    Lines7[76].X := 237.960; Lines7[76].Z := 284.913; Lines7[76].F := 800; Lines7[76].CMD := 1; Lines7[76].Param := 0; // G1 Linear [Op11 P1]
    Lines7[77].X := 237.085; Lines7[77].Z := 286.141; Lines7[77].F := 800; Lines7[77].CMD := 1; Lines7[77].Param := 0; // G1 Linear [Op11 P1]
    Lines7[78].X := 236.206; Lines7[78].Z := 287.367; Lines7[78].F := 800; Lines7[78].CMD := 1; Lines7[78].Param := 0; // G1 Linear [Op11 P1]
    Lines7[79].X := 235.321; Lines7[79].Z := 288.589; Lines7[79].F := 800; Lines7[79].CMD := 1; Lines7[79].Param := 0; // G1 Linear [Op11 P1]
    Lines7[80].X := 234.432; Lines7[80].Z := 289.808; Lines7[80].F := 800; Lines7[80].CMD := 1; Lines7[80].Param := 0; // G1 Linear [Op11 P1]
    Lines7[81].X := 233.539; Lines7[81].Z := 291.025; Lines7[81].F := 800; Lines7[81].CMD := 1; Lines7[81].Param := 0; // G1 Linear [Op11 P1]
    Lines7[82].X := 232.491; Lines7[82].Z := 292.440; Lines7[82].F := 800; Lines7[82].CMD := 1; Lines7[82].Param := 0; // G1 Linear [Op11 P1]
    Lines7[83].X := 231.587; Lines7[83].Z := 293.650; Lines7[83].F := 800; Lines7[83].CMD := 1; Lines7[83].Param := 0; // G1 Linear [Op11 P1]
    Lines7[84].X := 230.678; Lines7[84].Z := 294.858; Lines7[84].F := 800; Lines7[84].CMD := 1; Lines7[84].Param := 0; // G1 Linear [Op11 P1]
    Lines7[85].X := 229.765; Lines7[85].Z := 296.062; Lines7[85].F := 800; Lines7[85].CMD := 1; Lines7[85].Param := 0; // G1 Linear [Op11 P1]
    Lines7[86].X := 228.848; Lines7[86].Z := 297.263; Lines7[86].F := 800; Lines7[86].CMD := 1; Lines7[86].Param := 0; // G1 Linear [Op11 P1]
    Lines7[87].X := 227.925; Lines7[87].Z := 298.462; Lines7[87].F := 800; Lines7[87].CMD := 1; Lines7[87].Param := 0; // G1 Linear [Op11 P1]
    Lines7[88].X := 226.843; Lines7[88].Z := 299.857; Lines7[88].F := 800; Lines7[88].CMD := 1; Lines7[88].Param := 0; // G1 Linear [Op11 P1]
    Lines7[89].X := 225.911; Lines7[89].Z := 301.049; Lines7[89].F := 800; Lines7[89].CMD := 1; Lines7[89].Param := 0; // G1 Linear [Op11 P1]
    Lines7[90].X := 224.974; Lines7[90].Z := 302.238; Lines7[90].F := 800; Lines7[90].CMD := 1; Lines7[90].Param := 0; // G1 Linear [Op11 P1]
    Lines7[91].X := 224.032; Lines7[91].Z := 303.424; Lines7[91].F := 800; Lines7[91].CMD := 1; Lines7[91].Param := 0; // G1 Linear [Op11 P1]
    Lines7[92].X := 222.927; Lines7[92].Z := 304.805; Lines7[92].F := 800; Lines7[92].CMD := 1; Lines7[92].Param := 0; // G1 Linear [Op11 P1]
    Lines7[93].X := 212.927; Lines7[93].Z := 294.805; Lines7[93].F := 0; Lines7[93].CMD := 0; Lines7[93].Param := 0; // G0 Rapid [Op11 P1]
    Lines7[94].X := 212.927; Lines7[94].Z := 294.805; Lines7[94].F := 0; Lines7[94].CMD := 20; Lines7[94].Param := 80; // Spindle ON 800 RPM [Op11 P1]
    Lines7[95].X := 275.949; Lines7[95].Z := 196.000; Lines7[95].F := 0; Lines7[95].CMD := 0; Lines7[95].Param := 0; // G0 Rapid [Op12 P1]
    Lines7[96].X := 275.844; Lines7[96].Z := 227.468; Lines7[96].F := 800; Lines7[96].CMD := 1; Lines7[96].Param := 0; // G1 Linear [Op12 P1]
    Lines7[97].X := 275.813; Lines7[97].Z := 227.813; Lines7[97].F := 800; Lines7[97].CMD := 1; Lines7[97].Param := 0; // G1 Linear [Op12 P1]
    Lines7[98].X := 275.723; Lines7[98].Z := 228.147; Lines7[98].F := 800; Lines7[98].CMD := 1; Lines7[98].Param := 0; // G1 Linear [Op12 P1]
    Lines7[99].X := 275.576; Lines7[99].Z := 228.461; Lines7[99].F := 800; Lines7[99].CMD := 1; Lines7[99].Param := 0; // G1 Linear [Op12 P1]
    Lines8[0].X := 274.987; Lines8[0].Z := 229.860; Lines8[0].F := 800; Lines8[0].CMD := 1; Lines8[0].Param := 0; // G1 Linear [Op12 P1]
    Lines8[1].X := 274.392; Lines8[1].Z := 231.257; Lines8[1].F := 800; Lines8[1].CMD := 1; Lines8[1].Param := 0; // G1 Linear [Op12 P1]
    Lines8[2].X := 273.287; Lines8[2].Z := 233.809; Lines8[2].F := 800; Lines8[2].CMD := 1; Lines8[2].Param := 0; // G1 Linear [Op12 P1]
    Lines8[3].X := 272.677; Lines8[3].Z := 235.197; Lines8[3].F := 800; Lines8[3].CMD := 1; Lines8[3].Param := 0; // G1 Linear [Op12 P1]
    Lines8[4].X := 272.062; Lines8[4].Z := 236.582; Lines8[4].F := 800; Lines8[4].CMD := 1; Lines8[4].Param := 0; // G1 Linear [Op12 P1]
    Lines8[5].X := 271.441; Lines8[5].Z := 237.964; Lines8[5].F := 800; Lines8[5].CMD := 1; Lines8[5].Param := 0; // G1 Linear [Op12 P1]
    Lines8[6].X := 270.815; Lines8[6].Z := 239.343; Lines8[6].F := 800; Lines8[6].CMD := 1; Lines8[6].Param := 0; // G1 Linear [Op12 P1]
    Lines8[7].X := 269.654; Lines8[7].Z := 241.863; Lines8[7].F := 800; Lines8[7].CMD := 1; Lines8[7].Param := 0; // G1 Linear [Op12 P1]
    Lines8[8].X := 269.013; Lines8[8].Z := 243.233; Lines8[8].F := 800; Lines8[8].CMD := 1; Lines8[8].Param := 0; // G1 Linear [Op12 P1]
    Lines8[9].X := 268.367; Lines8[9].Z := 244.600; Lines8[9].F := 800; Lines8[9].CMD := 1; Lines8[9].Param := 0; // G1 Linear [Op12 P1]
    Lines8[10].X := 267.716; Lines8[10].Z := 245.964; Lines8[10].F := 800; Lines8[10].CMD := 1; Lines8[10].Param := 0; // G1 Linear [Op12 P1]
    Lines8[11].X := 267.059; Lines8[11].Z := 247.325; Lines8[11].F := 800; Lines8[11].CMD := 1; Lines8[11].Param := 0; // G1 Linear [Op12 P1]
    Lines8[12].X := 266.397; Lines8[12].Z := 248.683; Lines8[12].F := 800; Lines8[12].CMD := 1; Lines8[12].Param := 0; // G1 Linear [Op12 P1]
    Lines8[13].X := 265.729; Lines8[13].Z := 250.038; Lines8[13].F := 800; Lines8[13].CMD := 1; Lines8[13].Param := 0; // G1 Linear [Op12 P1]
    Lines8[14].X := 264.492; Lines8[14].Z := 252.514; Lines8[14].F := 800; Lines8[14].CMD := 1; Lines8[14].Param := 0; // G1 Linear [Op12 P1]
    Lines8[15].X := 263.810; Lines8[15].Z := 253.860; Lines8[15].F := 800; Lines8[15].CMD := 1; Lines8[15].Param := 0; // G1 Linear [Op12 P1]
    Lines8[16].X := 263.122; Lines8[16].Z := 255.203; Lines8[16].F := 800; Lines8[16].CMD := 1; Lines8[16].Param := 0; // G1 Linear [Op12 P1]
    Lines8[17].X := 262.429; Lines8[17].Z := 256.543; Lines8[17].F := 800; Lines8[17].CMD := 1; Lines8[17].Param := 0; // G1 Linear [Op12 P1]
    Lines8[18].X := 261.731; Lines8[18].Z := 257.880; Lines8[18].F := 800; Lines8[18].CMD := 1; Lines8[18].Param := 0; // G1 Linear [Op12 P1]
    Lines8[19].X := 261.027; Lines8[19].Z := 259.214; Lines8[19].F := 800; Lines8[19].CMD := 1; Lines8[19].Param := 0; // G1 Linear [Op12 P1]
    Lines8[20].X := 260.319; Lines8[20].Z := 260.545; Lines8[20].F := 800; Lines8[20].CMD := 1; Lines8[20].Param := 0; // G1 Linear [Op12 P1]
    Lines8[21].X := 259.005; Lines8[21].Z := 262.977; Lines8[21].F := 800; Lines8[21].CMD := 1; Lines8[21].Param := 0; // G1 Linear [Op12 P1]
    Lines8[22].X := 258.282; Lines8[22].Z := 264.300; Lines8[22].F := 800; Lines8[22].CMD := 1; Lines8[22].Param := 0; // G1 Linear [Op12 P1]
    Lines8[23].X := 257.552; Lines8[23].Z := 265.619; Lines8[23].F := 800; Lines8[23].CMD := 1; Lines8[23].Param := 0; // G1 Linear [Op12 P1]
    Lines8[24].X := 256.818; Lines8[24].Z := 266.935; Lines8[24].F := 800; Lines8[24].CMD := 1; Lines8[24].Param := 0; // G1 Linear [Op12 P1]
    Lines8[25].X := 256.078; Lines8[25].Z := 268.248; Lines8[25].F := 800; Lines8[25].CMD := 1; Lines8[25].Param := 0; // G1 Linear [Op12 P1]
    Lines8[26].X := 255.333; Lines8[26].Z := 269.558; Lines8[26].F := 800; Lines8[26].CMD := 1; Lines8[26].Param := 0; // G1 Linear [Op12 P1]
    Lines8[27].X := 254.583; Lines8[27].Z := 270.865; Lines8[27].F := 800; Lines8[27].CMD := 1; Lines8[27].Param := 0; // G1 Linear [Op12 P1]
    Lines8[28].X := 253.827; Lines8[28].Z := 272.169; Lines8[28].F := 800; Lines8[28].CMD := 1; Lines8[28].Param := 0; // G1 Linear [Op12 P1]
    Lines8[29].X := 253.067; Lines8[29].Z := 273.470; Lines8[29].F := 800; Lines8[29].CMD := 1; Lines8[29].Param := 0; // G1 Linear [Op12 P1]
    Lines8[30].X := 252.300; Lines8[30].Z := 274.768; Lines8[30].F := 800; Lines8[30].CMD := 1; Lines8[30].Param := 0; // G1 Linear [Op12 P1]
    Lines8[31].X := 251.529; Lines8[31].Z := 276.063; Lines8[31].F := 800; Lines8[31].CMD := 1; Lines8[31].Param := 0; // G1 Linear [Op12 P1]
    Lines8[32].X := 250.752; Lines8[32].Z := 277.355; Lines8[32].F := 800; Lines8[32].CMD := 1; Lines8[32].Param := 0; // G1 Linear [Op12 P1]
    Lines8[33].X := 249.970; Lines8[33].Z := 278.643; Lines8[33].F := 800; Lines8[33].CMD := 1; Lines8[33].Param := 0; // G1 Linear [Op12 P1]
    Lines8[34].X := 248.523; Lines8[34].Z := 280.998; Lines8[34].F := 800; Lines8[34].CMD := 1; Lines8[34].Param := 0; // G1 Linear [Op12 P1]
    Lines8[35].X := 247.057; Lines8[35].Z := 283.343; Lines8[35].F := 800; Lines8[35].CMD := 1; Lines8[35].Param := 0; // G1 Linear [Op12 P1]
    Lines8[36].X := 246.250; Lines8[36].Z := 284.617; Lines8[36].F := 800; Lines8[36].CMD := 1; Lines8[36].Param := 0; // G1 Linear [Op12 P1]
    Lines8[37].X := 245.438; Lines8[37].Z := 285.888; Lines8[37].F := 800; Lines8[37].CMD := 1; Lines8[37].Param := 0; // G1 Linear [Op12 P1]
    Lines8[38].X := 244.621; Lines8[38].Z := 287.157; Lines8[38].F := 800; Lines8[38].CMD := 1; Lines8[38].Param := 0; // G1 Linear [Op12 P1]
    Lines8[39].X := 243.798; Lines8[39].Z := 288.422; Lines8[39].F := 800; Lines8[39].CMD := 1; Lines8[39].Param := 0; // G1 Linear [Op12 P1]
    Lines8[40].X := 242.971; Lines8[40].Z := 289.684; Lines8[40].F := 800; Lines8[40].CMD := 1; Lines8[40].Param := 0; // G1 Linear [Op12 P1]
    Lines8[41].X := 242.137; Lines8[41].Z := 290.944; Lines8[41].F := 800; Lines8[41].CMD := 1; Lines8[41].Param := 0; // G1 Linear [Op12 P1]
    Lines8[42].X := 240.596; Lines8[42].Z := 293.244; Lines8[42].F := 800; Lines8[42].CMD := 1; Lines8[42].Param := 0; // G1 Linear [Op12 P1]
    Lines8[43].X := 239.748; Lines8[43].Z := 294.495; Lines8[43].F := 800; Lines8[43].CMD := 1; Lines8[43].Param := 0; // G1 Linear [Op12 P1]
    Lines8[44].X := 238.894; Lines8[44].Z := 295.742; Lines8[44].F := 800; Lines8[44].CMD := 1; Lines8[44].Param := 0; // G1 Linear [Op12 P1]
    Lines8[45].X := 238.035; Lines8[45].Z := 296.987; Lines8[45].F := 800; Lines8[45].CMD := 1; Lines8[45].Param := 0; // G1 Linear [Op12 P1]
    Lines8[46].X := 237.171; Lines8[46].Z := 298.228; Lines8[46].F := 800; Lines8[46].CMD := 1; Lines8[46].Param := 0; // G1 Linear [Op12 P1]
    Lines8[47].X := 236.302; Lines8[47].Z := 299.466; Lines8[47].F := 800; Lines8[47].CMD := 1; Lines8[47].Param := 0; // G1 Linear [Op12 P1]
    Lines8[48].X := 235.427; Lines8[48].Z := 300.702; Lines8[48].F := 800; Lines8[48].CMD := 1; Lines8[48].Param := 0; // G1 Linear [Op12 P1]
    Lines8[49].X := 234.547; Lines8[49].Z := 301.934; Lines8[49].F := 800; Lines8[49].CMD := 1; Lines8[49].Param := 0; // G1 Linear [Op12 P1]
    Lines8[50].X := 233.662; Lines8[50].Z := 303.163; Lines8[50].F := 800; Lines8[50].CMD := 1; Lines8[50].Param := 0; // G1 Linear [Op12 P1]
    Lines8[51].X := 232.025; Lines8[51].Z := 305.409; Lines8[51].F := 800; Lines8[51].CMD := 1; Lines8[51].Param := 0; // G1 Linear [Op12 P1]
    Lines8[52].X := 231.125; Lines8[52].Z := 306.629; Lines8[52].F := 800; Lines8[52].CMD := 1; Lines8[52].Param := 0; // G1 Linear [Op12 P1]
    Lines8[53].X := 230.219; Lines8[53].Z := 307.847; Lines8[53].F := 800; Lines8[53].CMD := 1; Lines8[53].Param := 0; // G1 Linear [Op12 P1]
    Lines8[54].X := 229.308; Lines8[54].Z := 309.061; Lines8[54].F := 800; Lines8[54].CMD := 1; Lines8[54].Param := 0; // G1 Linear [Op12 P1]
    Lines8[55].X := 228.392; Lines8[55].Z := 310.272; Lines8[55].F := 800; Lines8[55].CMD := 1; Lines8[55].Param := 0; // G1 Linear [Op12 P1]
    Lines8[56].X := 218.392; Lines8[56].Z := 300.272; Lines8[56].F := 0; Lines8[56].CMD := 0; Lines8[56].Param := 0; // G0 Rapid [Op12 P1]
    Lines8[57].X := 218.392; Lines8[57].Z := 300.272; Lines8[57].F := 0; Lines8[57].CMD := 20; Lines8[57].Param := 80; // Spindle ON 800 RPM [Op12 P1]
    Lines8[58].X := 275.949; Lines8[58].Z := 196.000; Lines8[58].F := 0; Lines8[58].CMD := 0; Lines8[58].Param := 0; // G0 Rapid [Op13 P1]
    Lines8[59].X := 275.819; Lines8[59].Z := 235.000; Lines8[59].F := 400; Lines8[59].CMD := 1; Lines8[59].Param := 0; // G1 Linear [Op13 P1]
    Lines8[60].X := 274.979; Lines8[60].Z := 237.394; Lines8[60].F := 400; Lines8[60].CMD := 1; Lines8[60].Param := 0; // G1 Linear [Op13 P1]
    Lines8[61].X := 274.552; Lines8[61].Z := 238.587; Lines8[61].F := 400; Lines8[61].CMD := 1; Lines8[61].Param := 0; // G1 Linear [Op13 P1]
    Lines8[62].X := 274.034; Lines8[62].Z := 240.016; Lines8[62].F := 400; Lines8[62].CMD := 1; Lines8[62].Param := 0; // G1 Linear [Op13 P1]
    Lines8[63].X := 273.597; Lines8[63].Z := 241.204; Lines8[63].F := 400; Lines8[63].CMD := 1; Lines8[63].Param := 0; // G1 Linear [Op13 P1]
    Lines8[64].X := 273.067; Lines8[64].Z := 242.627; Lines8[64].F := 400; Lines8[64].CMD := 1; Lines8[64].Param := 0; // G1 Linear [Op13 P1]
    Lines8[65].X := 272.621; Lines8[65].Z := 243.811; Lines8[65].F := 400; Lines8[65].CMD := 1; Lines8[65].Param := 0; // G1 Linear [Op13 P1]
    Lines8[66].X := 272.079; Lines8[66].Z := 245.228; Lines8[66].F := 400; Lines8[66].CMD := 1; Lines8[66].Param := 0; // G1 Linear [Op13 P1]
    Lines8[67].X := 271.623; Lines8[67].Z := 246.406; Lines8[67].F := 400; Lines8[67].CMD := 1; Lines8[67].Param := 0; // G1 Linear [Op13 P1]
    Lines8[68].X := 271.070; Lines8[68].Z := 247.817; Lines8[68].F := 400; Lines8[68].CMD := 1; Lines8[68].Param := 0; // G1 Linear [Op13 P1]
    Lines8[69].X := 270.510; Lines8[69].Z := 249.225; Lines8[69].F := 400; Lines8[69].CMD := 1; Lines8[69].Param := 0; // G1 Linear [Op13 P1]
    Lines8[70].X := 270.038; Lines8[70].Z := 250.396; Lines8[70].F := 400; Lines8[70].CMD := 1; Lines8[70].Param := 0; // G1 Linear [Op13 P1]
    Lines8[71].X := 269.563; Lines8[71].Z := 251.564; Lines8[71].F := 400; Lines8[71].CMD := 1; Lines8[71].Param := 0; // G1 Linear [Op13 P1]
    Lines8[72].X := 268.986; Lines8[72].Z := 252.963; Lines8[72].F := 400; Lines8[72].CMD := 1; Lines8[72].Param := 0; // G1 Linear [Op13 P1]
    Lines8[73].X := 268.010; Lines8[73].Z := 255.288; Lines8[73].F := 400; Lines8[73].CMD := 1; Lines8[73].Param := 0; // G1 Linear [Op13 P1]
    Lines8[74].X := 267.515; Lines8[74].Z := 256.447; Lines8[74].F := 400; Lines8[74].CMD := 1; Lines8[74].Param := 0; // G1 Linear [Op13 P1]
    Lines8[75].X := 266.915; Lines8[75].Z := 257.834; Lines8[75].F := 400; Lines8[75].CMD := 1; Lines8[75].Param := 0; // G1 Linear [Op13 P1]
    Lines8[76].X := 266.411; Lines8[76].Z := 258.988; Lines8[76].F := 400; Lines8[76].CMD := 1; Lines8[76].Param := 0; // G1 Linear [Op13 P1]
    Lines8[77].X := 265.800; Lines8[77].Z := 260.370; Lines8[77].F := 400; Lines8[77].CMD := 1; Lines8[77].Param := 0; // G1 Linear [Op13 P1]
    Lines8[78].X := 265.285; Lines8[78].Z := 261.518; Lines8[78].F := 400; Lines8[78].CMD := 1; Lines8[78].Param := 0; // G1 Linear [Op13 P1]
    Lines8[79].X := 264.662; Lines8[79].Z := 262.894; Lines8[79].F := 400; Lines8[79].CMD := 1; Lines8[79].Param := 0; // G1 Linear [Op13 P1]
    Lines8[80].X := 264.033; Lines8[80].Z := 264.266; Lines8[80].F := 400; Lines8[80].CMD := 1; Lines8[80].Param := 0; // G1 Linear [Op13 P1]
    Lines8[81].X := 263.503; Lines8[81].Z := 265.408; Lines8[81].F := 400; Lines8[81].CMD := 1; Lines8[81].Param := 0; // G1 Linear [Op13 P1]
    Lines8[82].X := 262.969; Lines8[82].Z := 266.546; Lines8[82].F := 400; Lines8[82].CMD := 1; Lines8[82].Param := 0; // G1 Linear [Op13 P1]
    Lines8[83].X := 262.322; Lines8[83].Z := 267.910; Lines8[83].F := 400; Lines8[83].CMD := 1; Lines8[83].Param := 0; // G1 Linear [Op13 P1]
    Lines8[84].X := 261.779; Lines8[84].Z := 269.044; Lines8[84].F := 400; Lines8[84].CMD := 1; Lines8[84].Param := 0; // G1 Linear [Op13 P1]
    Lines8[85].X := 261.120; Lines8[85].Z := 270.401; Lines8[85].F := 400; Lines8[85].CMD := 1; Lines8[85].Param := 0; // G1 Linear [Op13 P1]
    Lines8[86].X := 260.008; Lines8[86].Z := 272.657; Lines8[86].F := 400; Lines8[86].CMD := 1; Lines8[86].Param := 0; // G1 Linear [Op13 P1]
    Lines8[87].X := 259.446; Lines8[87].Z := 273.781; Lines8[87].F := 400; Lines8[87].CMD := 1; Lines8[87].Param := 0; // G1 Linear [Op13 P1]
    Lines8[88].X := 258.765; Lines8[88].Z := 275.127; Lines8[88].F := 400; Lines8[88].CMD := 1; Lines8[88].Param := 0; // G1 Linear [Op13 P1]
    Lines8[89].X := 257.616; Lines8[89].Z := 277.364; Lines8[89].F := 400; Lines8[89].CMD := 1; Lines8[89].Param := 0; // G1 Linear [Op13 P1]
    Lines8[90].X := 257.034; Lines8[90].Z := 278.478; Lines8[90].F := 400; Lines8[90].CMD := 1; Lines8[90].Param := 0; // G1 Linear [Op13 P1]
    Lines8[91].X := 256.331; Lines8[91].Z := 279.813; Lines8[91].F := 400; Lines8[91].CMD := 1; Lines8[91].Param := 0; // G1 Linear [Op13 P1]
    Lines8[92].X := 255.621; Lines8[92].Z := 281.144; Lines8[92].F := 400; Lines8[92].CMD := 1; Lines8[92].Param := 0; // G1 Linear [Op13 P1]
    Lines8[93].X := 255.024; Lines8[93].Z := 282.251; Lines8[93].F := 400; Lines8[93].CMD := 1; Lines8[93].Param := 0; // G1 Linear [Op13 P1]
    Lines8[94].X := 254.423; Lines8[94].Z := 283.356; Lines8[94].F := 400; Lines8[94].CMD := 1; Lines8[94].Param := 0; // G1 Linear [Op13 P1]
    Lines8[95].X := 253.696; Lines8[95].Z := 284.679; Lines8[95].F := 400; Lines8[95].CMD := 1; Lines8[95].Param := 0; // G1 Linear [Op13 P1]
    Lines8[96].X := 252.470; Lines8[96].Z := 286.876; Lines8[96].F := 400; Lines8[96].CMD := 1; Lines8[96].Param := 0; // G1 Linear [Op13 P1]
    Lines8[97].X := 251.726; Lines8[97].Z := 288.190; Lines8[97].F := 400; Lines8[97].CMD := 1; Lines8[97].Param := 0; // G1 Linear [Op13 P1]
    Lines8[98].X := 251.101; Lines8[98].Z := 289.282; Lines8[98].F := 400; Lines8[98].CMD := 1; Lines8[98].Param := 0; // G1 Linear [Op13 P1]
    Lines8[99].X := 250.471; Lines8[99].Z := 290.373; Lines8[99].F := 400; Lines8[99].CMD := 1; Lines8[99].Param := 0; // G1 Linear [Op13 P1]
    Lines9[0].X := 249.710; Lines9[0].Z := 291.678; Lines9[0].F := 400; Lines9[0].CMD := 1; Lines9[0].Param := 0; // G1 Linear [Op13 P1]
    Lines9[1].X := 249.071; Lines9[1].Z := 292.763; Lines9[1].F := 400; Lines9[1].CMD := 1; Lines9[1].Param := 0; // G1 Linear [Op13 P1]
    Lines9[2].X := 248.297; Lines9[2].Z := 294.062; Lines9[2].F := 400; Lines9[2].CMD := 1; Lines9[2].Param := 0; // G1 Linear [Op13 P1]
    Lines9[3].X := 246.995; Lines9[3].Z := 296.220; Lines9[3].F := 400; Lines9[3].CMD := 1; Lines9[3].Param := 0; // G1 Linear [Op13 P1]
    Lines9[4].X := 246.336; Lines9[4].Z := 297.296; Lines9[4].F := 400; Lines9[4].CMD := 1; Lines9[4].Param := 0; // G1 Linear [Op13 P1]
    Lines9[5].X := 245.541; Lines9[5].Z := 298.584; Lines9[5].F := 400; Lines9[5].CMD := 1; Lines9[5].Param := 0; // G1 Linear [Op13 P1]
    Lines9[6].X := 244.873; Lines9[6].Z := 299.654; Lines9[6].F := 400; Lines9[6].CMD := 1; Lines9[6].Param := 0; // G1 Linear [Op13 P1]
    Lines9[7].X := 244.065; Lines9[7].Z := 300.936; Lines9[7].F := 400; Lines9[7].CMD := 1; Lines9[7].Param := 0; // G1 Linear [Op13 P1]
    Lines9[8].X := 243.387; Lines9[8].Z := 302.002; Lines9[8].F := 400; Lines9[8].CMD := 1; Lines9[8].Param := 0; // G1 Linear [Op13 P1]
    Lines9[9].X := 242.568; Lines9[9].Z := 303.278; Lines9[9].F := 400; Lines9[9].CMD := 1; Lines9[9].Param := 0; // G1 Linear [Op13 P1]
    Lines9[10].X := 241.881; Lines9[10].Z := 304.338; Lines9[10].F := 400; Lines9[10].CMD := 1; Lines9[10].Param := 0; // G1 Linear [Op13 P1]
    Lines9[11].X := 241.049; Lines9[11].Z := 305.608; Lines9[11].F := 400; Lines9[11].CMD := 1; Lines9[11].Param := 0; // G1 Linear [Op13 P1]
    Lines9[12].X := 240.352; Lines9[12].Z := 306.664; Lines9[12].F := 400; Lines9[12].CMD := 1; Lines9[12].Param := 0; // G1 Linear [Op13 P1]
    Lines9[13].X := 239.509; Lines9[13].Z := 307.927; Lines9[13].F := 400; Lines9[13].CMD := 1; Lines9[13].Param := 0; // G1 Linear [Op13 P1]
    Lines9[14].X := 238.802; Lines9[14].Z := 308.978; Lines9[14].F := 400; Lines9[14].CMD := 1; Lines9[14].Param := 0; // G1 Linear [Op13 P1]
    Lines9[15].X := 237.947; Lines9[15].Z := 310.236; Lines9[15].F := 400; Lines9[15].CMD := 1; Lines9[15].Param := 0; // G1 Linear [Op13 P1]
    Lines9[16].X := 237.230; Lines9[16].Z := 311.281; Lines9[16].F := 400; Lines9[16].CMD := 1; Lines9[16].Param := 0; // G1 Linear [Op13 P1]
    Lines9[17].X := 236.364; Lines9[17].Z := 312.533; Lines9[17].F := 400; Lines9[17].CMD := 1; Lines9[17].Param := 0; // G1 Linear [Op13 P1]
    Lines9[18].X := 226.364; Lines9[18].Z := 302.533; Lines9[18].F := 0; Lines9[18].CMD := 0; Lines9[18].Param := 0; // G0 Rapid [Op13 P1]
    Lines9[19].X := 226.364; Lines9[19].Z := 302.533; Lines9[19].F := 0; Lines9[19].CMD := 20; Lines9[19].Param := 80; // Spindle ON 800 RPM [Op13 P1]
    Lines9[20].X := 275.882; Lines9[20].Z := 216.000; Lines9[20].F := 0; Lines9[20].CMD := 0; Lines9[20].Param := 0; // G0 Rapid [Op14 P1]
    Lines9[21].X := 275.799; Lines9[21].Z := 241.000; Lines9[21].F := 400; Lines9[21].CMD := 1; Lines9[21].Param := 0; // G1 Linear [Op14 P1]
    Lines9[22].X := 275.441; Lines9[22].Z := 242.217; Lines9[22].F := 400; Lines9[22].CMD := 1; Lines9[22].Param := 0; // G1 Linear [Op14 P1]
    Lines9[23].X := 275.077; Lines9[23].Z := 243.432; Lines9[23].F := 400; Lines9[23].CMD := 1; Lines9[23].Param := 0; // G1 Linear [Op14 P1]
    Lines9[24].X := 274.409; Lines9[24].Z := 245.611; Lines9[24].F := 400; Lines9[24].CMD := 1; Lines9[24].Param := 0; // G1 Linear [Op14 P1]
    Lines9[25].X := 274.030; Lines9[25].Z := 246.818; Lines9[25].F := 400; Lines9[25].CMD := 1; Lines9[25].Param := 0; // G1 Linear [Op14 P1]
    Lines9[26].X := 273.645; Lines9[26].Z := 248.023; Lines9[26].F := 400; Lines9[26].CMD := 1; Lines9[26].Param := 0; // G1 Linear [Op14 P1]
    Lines9[27].X := 273.255; Lines9[27].Z := 249.225; Lines9[27].F := 400; Lines9[27].CMD := 1; Lines9[27].Param := 0; // G1 Linear [Op14 P1]
    Lines9[28].X := 272.859; Lines9[28].Z := 250.424; Lines9[28].F := 400; Lines9[28].CMD := 1; Lines9[28].Param := 0; // G1 Linear [Op14 P1]
    Lines9[29].X := 272.132; Lines9[29].Z := 252.576; Lines9[29].F := 400; Lines9[29].CMD := 1; Lines9[29].Param := 0; // G1 Linear [Op14 P1]
    Lines9[30].X := 271.720; Lines9[30].Z := 253.768; Lines9[30].F := 400; Lines9[30].CMD := 1; Lines9[30].Param := 0; // G1 Linear [Op14 P1]
    Lines9[31].X := 271.303; Lines9[31].Z := 254.958; Lines9[31].F := 400; Lines9[31].CMD := 1; Lines9[31].Param := 0; // G1 Linear [Op14 P1]
    Lines9[32].X := 270.880; Lines9[32].Z := 256.145; Lines9[32].F := 400; Lines9[32].CMD := 1; Lines9[32].Param := 0; // G1 Linear [Op14 P1]
    Lines9[33].X := 270.452; Lines9[33].Z := 257.329; Lines9[33].F := 400; Lines9[33].CMD := 1; Lines9[33].Param := 0; // G1 Linear [Op14 P1]
    Lines9[34].X := 270.018; Lines9[34].Z := 258.511; Lines9[34].F := 400; Lines9[34].CMD := 1; Lines9[34].Param := 0; // G1 Linear [Op14 P1]
    Lines9[35].X := 269.579; Lines9[35].Z := 259.690; Lines9[35].F := 400; Lines9[35].CMD := 1; Lines9[35].Param := 0; // G1 Linear [Op14 P1]
    Lines9[36].X := 268.773; Lines9[36].Z := 261.806; Lines9[36].F := 400; Lines9[36].CMD := 1; Lines9[36].Param := 0; // G1 Linear [Op14 P1]
    Lines9[37].X := 268.318; Lines9[37].Z := 262.977; Lines9[37].F := 400; Lines9[37].CMD := 1; Lines9[37].Param := 0; // G1 Linear [Op14 P1]
    Lines9[38].X := 267.858; Lines9[38].Z := 264.147; Lines9[38].F := 400; Lines9[38].CMD := 1; Lines9[38].Param := 0; // G1 Linear [Op14 P1]
    Lines9[39].X := 267.391; Lines9[39].Z := 265.313; Lines9[39].F := 400; Lines9[39].CMD := 1; Lines9[39].Param := 0; // G1 Linear [Op14 P1]
    Lines9[40].X := 266.919; Lines9[40].Z := 266.477; Lines9[40].F := 400; Lines9[40].CMD := 1; Lines9[40].Param := 0; // G1 Linear [Op14 P1]
    Lines9[41].X := 266.442; Lines9[41].Z := 267.639; Lines9[41].F := 400; Lines9[41].CMD := 1; Lines9[41].Param := 0; // G1 Linear [Op14 P1]
    Lines9[42].X := 265.959; Lines9[42].Z := 268.797; Lines9[42].F := 400; Lines9[42].CMD := 1; Lines9[42].Param := 0; // G1 Linear [Op14 P1]
    Lines9[43].X := 265.075; Lines9[43].Z := 270.877; Lines9[43].F := 400; Lines9[43].CMD := 1; Lines9[43].Param := 0; // G1 Linear [Op14 P1]
    Lines9[44].X := 264.576; Lines9[44].Z := 272.028; Lines9[44].F := 400; Lines9[44].CMD := 1; Lines9[44].Param := 0; // G1 Linear [Op14 P1]
    Lines9[45].X := 264.072; Lines9[45].Z := 273.177; Lines9[45].F := 400; Lines9[45].CMD := 1; Lines9[45].Param := 0; // G1 Linear [Op14 P1]
    Lines9[46].X := 263.562; Lines9[46].Z := 274.323; Lines9[46].F := 400; Lines9[46].CMD := 1; Lines9[46].Param := 0; // G1 Linear [Op14 P1]
    Lines9[47].X := 263.047; Lines9[47].Z := 275.467; Lines9[47].F := 400; Lines9[47].CMD := 1; Lines9[47].Param := 0; // G1 Linear [Op14 P1]
    Lines9[48].X := 262.525; Lines9[48].Z := 276.608; Lines9[48].F := 400; Lines9[48].CMD := 1; Lines9[48].Param := 0; // G1 Linear [Op14 P1]
    Lines9[49].X := 261.999; Lines9[49].Z := 277.747; Lines9[49].F := 400; Lines9[49].CMD := 1; Lines9[49].Param := 0; // G1 Linear [Op14 P1]
    Lines9[50].X := 261.037; Lines9[50].Z := 279.789; Lines9[50].F := 400; Lines9[50].CMD := 1; Lines9[50].Param := 0; // G1 Linear [Op14 P1]
    Lines9[51].X := 260.494; Lines9[51].Z := 280.920; Lines9[51].F := 400; Lines9[51].CMD := 1; Lines9[51].Param := 0; // G1 Linear [Op14 P1]
    Lines9[52].X := 259.946; Lines9[52].Z := 282.049; Lines9[52].F := 400; Lines9[52].CMD := 1; Lines9[52].Param := 0; // G1 Linear [Op14 P1]
    Lines9[53].X := 259.393; Lines9[53].Z := 283.175; Lines9[53].F := 400; Lines9[53].CMD := 1; Lines9[53].Param := 0; // G1 Linear [Op14 P1]
    Lines9[54].X := 258.834; Lines9[54].Z := 284.298; Lines9[54].F := 400; Lines9[54].CMD := 1; Lines9[54].Param := 0; // G1 Linear [Op14 P1]
    Lines9[55].X := 258.269; Lines9[55].Z := 285.419; Lines9[55].F := 400; Lines9[55].CMD := 1; Lines9[55].Param := 0; // G1 Linear [Op14 P1]
    Lines9[56].X := 257.699; Lines9[56].Z := 286.537; Lines9[56].F := 400; Lines9[56].CMD := 1; Lines9[56].Param := 0; // G1 Linear [Op14 P1]
    Lines9[57].X := 257.123; Lines9[57].Z := 287.653; Lines9[57].F := 400; Lines9[57].CMD := 1; Lines9[57].Param := 0; // G1 Linear [Op14 P1]
    Lines9[58].X := 256.542; Lines9[58].Z := 288.766; Lines9[58].F := 400; Lines9[58].CMD := 1; Lines9[58].Param := 0; // G1 Linear [Op14 P1]
    Lines9[59].X := 255.481; Lines9[59].Z := 290.763; Lines9[59].F := 400; Lines9[59].CMD := 1; Lines9[59].Param := 0; // G1 Linear [Op14 P1]
    Lines9[60].X := 254.884; Lines9[60].Z := 291.869; Lines9[60].F := 400; Lines9[60].CMD := 1; Lines9[60].Param := 0; // G1 Linear [Op14 P1]
    Lines9[61].X := 254.281; Lines9[61].Z := 292.972; Lines9[61].F := 400; Lines9[61].CMD := 1; Lines9[61].Param := 0; // G1 Linear [Op14 P1]
    Lines9[62].X := 253.673; Lines9[62].Z := 294.072; Lines9[62].F := 400; Lines9[62].CMD := 1; Lines9[62].Param := 0; // G1 Linear [Op14 P1]
    Lines9[63].X := 253.059; Lines9[63].Z := 295.170; Lines9[63].F := 400; Lines9[63].CMD := 1; Lines9[63].Param := 0; // G1 Linear [Op14 P1]
    Lines9[64].X := 251.940; Lines9[64].Z := 297.140; Lines9[64].F := 400; Lines9[64].CMD := 1; Lines9[64].Param := 0; // G1 Linear [Op14 P1]
    Lines9[65].X := 251.310; Lines9[65].Z := 298.230; Lines9[65].F := 400; Lines9[65].CMD := 1; Lines9[65].Param := 0; // G1 Linear [Op14 P1]
    Lines9[66].X := 250.675; Lines9[66].Z := 299.318; Lines9[66].F := 400; Lines9[66].CMD := 1; Lines9[66].Param := 0; // G1 Linear [Op14 P1]
    Lines9[67].X := 250.035; Lines9[67].Z := 300.404; Lines9[67].F := 400; Lines9[67].CMD := 1; Lines9[67].Param := 0; // G1 Linear [Op14 P1]
    Lines9[68].X := 249.388; Lines9[68].Z := 301.487; Lines9[68].F := 400; Lines9[68].CMD := 1; Lines9[68].Param := 0; // G1 Linear [Op14 P1]
    Lines9[69].X := 248.737; Lines9[69].Z := 302.567; Lines9[69].F := 400; Lines9[69].CMD := 1; Lines9[69].Param := 0; // G1 Linear [Op14 P1]
    Lines9[70].X := 248.079; Lines9[70].Z := 303.644; Lines9[70].F := 400; Lines9[70].CMD := 1; Lines9[70].Param := 0; // G1 Linear [Op14 P1]
    Lines9[71].X := 246.882; Lines9[71].Z := 305.578; Lines9[71].F := 400; Lines9[71].CMD := 1; Lines9[71].Param := 0; // G1 Linear [Op14 P1]
    Lines9[72].X := 246.209; Lines9[72].Z := 306.648; Lines9[72].F := 400; Lines9[72].CMD := 1; Lines9[72].Param := 0; // G1 Linear [Op14 P1]
    Lines9[73].X := 245.530; Lines9[73].Z := 307.716; Lines9[73].F := 400; Lines9[73].CMD := 1; Lines9[73].Param := 0; // G1 Linear [Op14 P1]
    Lines9[74].X := 244.846; Lines9[74].Z := 308.781; Lines9[74].F := 400; Lines9[74].CMD := 1; Lines9[74].Param := 0; // G1 Linear [Op14 P1]
    Lines9[75].X := 244.156; Lines9[75].Z := 309.843; Lines9[75].F := 400; Lines9[75].CMD := 1; Lines9[75].Param := 0; // G1 Linear [Op14 P1]
    Lines9[76].X := 243.460; Lines9[76].Z := 310.903; Lines9[76].F := 400; Lines9[76].CMD := 1; Lines9[76].Param := 0; // G1 Linear [Op14 P1]
    Lines9[77].X := 242.759; Lines9[77].Z := 311.961; Lines9[77].F := 400; Lines9[77].CMD := 1; Lines9[77].Param := 0; // G1 Linear [Op14 P1]
    Lines9[78].X := 232.759; Lines9[78].Z := 301.961; Lines9[78].F := 0; Lines9[78].CMD := 0; Lines9[78].Param := 0; // G0 Rapid [Op14 P1]
    Lines9[79].X := 232.759; Lines9[79].Z := 301.961; Lines9[79].F := 0; Lines9[79].CMD := 20; Lines9[79].Param := 80; // Spindle ON 800 RPM [Op14 P1]
    Lines9[80].X := 275.865; Lines9[80].Z := 221.000; Lines9[80].F := 0; Lines9[80].CMD := 0; Lines9[80].Param := 0; // G0 Rapid [Op15 P1]
    Lines9[81].X := 275.772; Lines9[81].Z := 249.000; Lines9[81].F := 400; Lines9[81].CMD := 1; Lines9[81].Param := 0; // G1 Linear [Op15 P1]
    Lines9[82].X := 275.480; Lines9[82].Z := 250.242; Lines9[82].F := 400; Lines9[82].CMD := 1; Lines9[82].Param := 0; // G1 Linear [Op15 P1]
    Lines9[83].X := 275.240; Lines9[83].Z := 251.233; Lines9[83].F := 400; Lines9[83].CMD := 1; Lines9[83].Param := 0; // G1 Linear [Op15 P1]
    Lines9[84].X := 274.747; Lines9[84].Z := 253.209; Lines9[84].F := 400; Lines9[84].CMD := 1; Lines9[84].Param := 0; // G1 Linear [Op15 P1]
    Lines9[85].X := 274.235; Lines9[85].Z := 255.178; Lines9[85].F := 400; Lines9[85].CMD := 1; Lines9[85].Param := 0; // G1 Linear [Op15 P1]
    Lines9[86].X := 273.972; Lines9[86].Z := 256.159; Lines9[86].F := 400; Lines9[86].CMD := 1; Lines9[86].Param := 0; // G1 Linear [Op15 P1]
    Lines9[87].X := 273.637; Lines9[87].Z := 257.383; Lines9[87].F := 400; Lines9[87].CMD := 1; Lines9[87].Param := 0; // G1 Linear [Op15 P1]
    Lines9[88].X := 273.085; Lines9[88].Z := 259.334; Lines9[88].F := 400; Lines9[88].CMD := 1; Lines9[88].Param := 0; // G1 Linear [Op15 P1]
    Lines9[89].X := 272.802; Lines9[89].Z := 260.307; Lines9[89].F := 400; Lines9[89].CMD := 1; Lines9[89].Param := 0; // G1 Linear [Op15 P1]
    Lines9[90].X := 272.442; Lines9[90].Z := 261.520; Lines9[90].F := 400; Lines9[90].CMD := 1; Lines9[90].Param := 0; // G1 Linear [Op15 P1]
    Lines9[91].X := 272.148; Lines9[91].Z := 262.488; Lines9[91].F := 400; Lines9[91].CMD := 1; Lines9[91].Param := 0; // G1 Linear [Op15 P1]
    Lines9[92].X := 271.775; Lines9[92].Z := 263.696; Lines9[92].F := 400; Lines9[92].CMD := 1; Lines9[92].Param := 0; // G1 Linear [Op15 P1]
    Lines9[93].X := 271.162; Lines9[93].Z := 265.621; Lines9[93].F := 400; Lines9[93].CMD := 1; Lines9[93].Param := 0; // G1 Linear [Op15 P1]
    Lines9[94].X := 270.530; Lines9[94].Z := 267.539; Lines9[94].F := 400; Lines9[94].CMD := 1; Lines9[94].Param := 0; // G1 Linear [Op15 P1]
    Lines9[95].X := 270.125; Lines9[95].Z := 268.733; Lines9[95].F := 400; Lines9[95].CMD := 1; Lines9[95].Param := 0; // G1 Linear [Op15 P1]
    Lines9[96].X := 269.796; Lines9[96].Z := 269.686; Lines9[96].F := 400; Lines9[96].CMD := 1; Lines9[96].Param := 0; // G1 Linear [Op15 P1]
    Lines9[97].X := 269.125; Lines9[97].Z := 271.587; Lines9[97].F := 400; Lines9[97].CMD := 1; Lines9[97].Param := 0; // G1 Linear [Op15 P1]
    Lines9[98].X := 268.781; Lines9[98].Z := 272.534; Lines9[98].F := 400; Lines9[98].CMD := 1; Lines9[98].Param := 0; // G1 Linear [Op15 P1]
    Lines9[99].X := 268.346; Lines9[99].Z := 273.715; Lines9[99].F := 400; Lines9[99].CMD := 1; Lines9[99].Param := 0; // G1 Linear [Op15 P1]
    Lines10[0].X := 267.634; Lines10[0].Z := 275.599; Lines10[0].F := 400; Lines10[0].CMD := 1; Lines10[0].Param := 0; // G1 Linear [Op15 P1]
    Lines10[1].X := 267.271; Lines10[1].Z := 276.538; Lines10[1].F := 400; Lines10[1].CMD := 1; Lines10[1].Param := 0; // G1 Linear [Op15 P1]
    Lines10[2].X := 266.811; Lines10[2].Z := 277.708; Lines10[2].F := 400; Lines10[2].CMD := 1; Lines10[2].Param := 0; // G1 Linear [Op15 P1]
    Lines10[3].X := 266.437; Lines10[3].Z := 278.643; Lines10[3].F := 400; Lines10[3].CMD := 1; Lines10[3].Param := 0; // G1 Linear [Op15 P1]
    Lines10[4].X := 265.963; Lines10[4].Z := 279.808; Lines10[4].F := 400; Lines10[4].CMD := 1; Lines10[4].Param := 0; // G1 Linear [Op15 P1]
    Lines10[5].X := 265.482; Lines10[5].Z := 280.970; Lines10[5].F := 400; Lines10[5].CMD := 1; Lines10[5].Param := 0; // G1 Linear [Op15 P1]
    Lines10[6].X := 265.092; Lines10[6].Z := 281.897; Lines10[6].F := 400; Lines10[6].CMD := 1; Lines10[6].Param := 0; // G1 Linear [Op15 P1]
    Lines10[7].X := 264.298; Lines10[7].Z := 283.746; Lines10[7].F := 400; Lines10[7].CMD := 1; Lines10[7].Param := 0; // G1 Linear [Op15 P1]
    Lines10[8].X := 263.894; Lines10[8].Z := 284.667; Lines10[8].F := 400; Lines10[8].CMD := 1; Lines10[8].Param := 0; // G1 Linear [Op15 P1]
    Lines10[9].X := 263.382; Lines10[9].Z := 285.816; Lines10[9].F := 400; Lines10[9].CMD := 1; Lines10[9].Param := 0; // G1 Linear [Op15 P1]
    Lines10[10].X := 262.862; Lines10[10].Z := 286.962; Lines10[10].F := 400; Lines10[10].CMD := 1; Lines10[10].Param := 0; // G1 Linear [Op15 P1]
    Lines10[11].X := 262.442; Lines10[11].Z := 287.876; Lines10[11].F := 400; Lines10[11].CMD := 1; Lines10[11].Param := 0; // G1 Linear [Op15 P1]
    Lines10[12].X := 261.586; Lines10[12].Z := 289.699; Lines10[12].F := 400; Lines10[12].CMD := 1; Lines10[12].Param := 0; // G1 Linear [Op15 P1]
    Lines10[13].X := 260.712; Lines10[13].Z := 291.514; Lines10[13].F := 400; Lines10[13].CMD := 1; Lines10[13].Param := 0; // G1 Linear [Op15 P1]
    Lines10[14].X := 260.267; Lines10[14].Z := 292.418; Lines10[14].F := 400; Lines10[14].CMD := 1; Lines10[14].Param := 0; // G1 Linear [Op15 P1]
    Lines10[15].X := 259.705; Lines10[15].Z := 293.546; Lines10[15].F := 400; Lines10[15].CMD := 1; Lines10[15].Param := 0; // G1 Linear [Op15 P1]
    Lines10[16].X := 258.791; Lines10[16].Z := 295.343; Lines10[16].F := 400; Lines10[16].CMD := 1; Lines10[16].Param := 0; // G1 Linear [Op15 P1]
    Lines10[17].X := 258.327; Lines10[17].Z := 296.239; Lines10[17].F := 400; Lines10[17].CMD := 1; Lines10[17].Param := 0; // G1 Linear [Op15 P1]
    Lines10[18].X := 257.740; Lines10[18].Z := 297.356; Lines10[18].F := 400; Lines10[18].CMD := 1; Lines10[18].Param := 0; // G1 Linear [Op15 P1]
    Lines10[19].X := 256.785; Lines10[19].Z := 299.137; Lines10[19].F := 400; Lines10[19].CMD := 1; Lines10[19].Param := 0; // G1 Linear [Op15 P1]
    Lines10[20].X := 256.301; Lines10[20].Z := 300.025; Lines10[20].F := 400; Lines10[20].CMD := 1; Lines10[20].Param := 0; // G1 Linear [Op15 P1]
    Lines10[21].X := 255.689; Lines10[21].Z := 301.131; Lines10[21].F := 400; Lines10[21].CMD := 1; Lines10[21].Param := 0; // G1 Linear [Op15 P1]
    Lines10[22].X := 255.194; Lines10[22].Z := 302.014; Lines10[22].F := 400; Lines10[22].CMD := 1; Lines10[22].Param := 0; // G1 Linear [Op15 P1]
    Lines10[23].X := 254.569; Lines10[23].Z := 303.115; Lines10[23].F := 400; Lines10[23].CMD := 1; Lines10[23].Param := 0; // G1 Linear [Op15 P1]
    Lines10[24].X := 253.553; Lines10[24].Z := 304.870; Lines10[24].F := 400; Lines10[24].CMD := 1; Lines10[24].Param := 0; // G1 Linear [Op15 P1]
    Lines10[25].X := 252.518; Lines10[25].Z := 306.617; Lines10[25].F := 400; Lines10[25].CMD := 1; Lines10[25].Param := 0; // G1 Linear [Op15 P1]
    Lines10[26].X := 251.994; Lines10[26].Z := 307.487; Lines10[26].F := 400; Lines10[26].CMD := 1; Lines10[26].Param := 0; // G1 Linear [Op15 P1]
    Lines10[27].X := 251.332; Lines10[27].Z := 308.572; Lines10[27].F := 400; Lines10[27].CMD := 1; Lines10[27].Param := 0; // G1 Linear [Op15 P1]
    Lines10[28].X := 250.797; Lines10[28].Z := 309.438; Lines10[28].F := 400; Lines10[28].CMD := 1; Lines10[28].Param := 0; // G1 Linear [Op15 P1]
    Lines10[29].X := 250.122; Lines10[29].Z := 310.518; Lines10[29].F := 400; Lines10[29].CMD := 1; Lines10[29].Param := 0; // G1 Linear [Op15 P1]
    Lines10[30].X := 249.576; Lines10[30].Z := 311.380; Lines10[30].F := 400; Lines10[30].CMD := 1; Lines10[30].Param := 0; // G1 Linear [Op15 P1]
    Lines10[31].X := 248.888; Lines10[31].Z := 312.454; Lines10[31].F := 400; Lines10[31].CMD := 1; Lines10[31].Param := 0; // G1 Linear [Op15 P1]
    Lines10[32].X := 238.888; Lines10[32].Z := 302.454; Lines10[32].F := 0; Lines10[32].CMD := 0; Lines10[32].Param := 0; // G0 Rapid [Op15 P1]
    Lines10[33].X := 238.888; Lines10[33].Z := 302.454; Lines10[33].F := 0; Lines10[33].CMD := 20; Lines10[33].Param := 80; // Spindle ON 800 RPM [Op15 P1]
    Lines10[34].X := 275.866; Lines10[34].Z := 221.000; Lines10[34].F := 0; Lines10[34].CMD := 0; Lines10[34].Param := 0; // G0 Rapid [Op16 P1]
    Lines10[35].X := 275.749; Lines10[35].Z := 256.000; Lines10[35].F := 400; Lines10[35].CMD := 1; Lines10[35].Param := 0; // G1 Linear [Op16 P1]
    Lines10[36].X := 275.448; Lines10[36].Z := 257.769; Lines10[36].F := 400; Lines10[36].CMD := 1; Lines10[36].Param := 0; // G1 Linear [Op16 P1]
    Lines10[37].X := 275.126; Lines10[37].Z := 259.529; Lines10[37].F := 400; Lines10[37].CMD := 1; Lines10[37].Param := 0; // G1 Linear [Op16 P1]
    Lines10[38].X := 274.784; Lines10[38].Z := 261.282; Lines10[38].F := 400; Lines10[38].CMD := 1; Lines10[38].Param := 0; // G1 Linear [Op16 P1]
    Lines10[39].X := 274.579; Lines10[39].Z := 262.281; Lines10[39].F := 400; Lines10[39].CMD := 1; Lines10[39].Param := 0; // G1 Linear [Op16 P1]
    Lines10[40].X := 274.368; Lines10[40].Z := 263.276; Lines10[40].F := 400; Lines10[40].CMD := 1; Lines10[40].Param := 0; // G1 Linear [Op16 P1]
    Lines10[41].X := 273.982; Lines10[41].Z := 265.012; Lines10[41].F := 400; Lines10[41].CMD := 1; Lines10[41].Param := 0; // G1 Linear [Op16 P1]
    Lines10[42].X := 273.752; Lines10[42].Z := 266.001; Lines10[42].F := 400; Lines10[42].CMD := 1; Lines10[42].Param := 0; // G1 Linear [Op16 P1]
    Lines10[43].X := 273.516; Lines10[43].Z := 266.987; Lines10[43].F := 400; Lines10[43].CMD := 1; Lines10[43].Param := 0; // G1 Linear [Op16 P1]
    Lines10[44].X := 273.273; Lines10[44].Z := 267.971; Lines10[44].F := 400; Lines10[44].CMD := 1; Lines10[44].Param := 0; // G1 Linear [Op16 P1]
    Lines10[45].X := 273.087; Lines10[45].Z := 268.707; Lines10[45].F := 400; Lines10[45].CMD := 1; Lines10[45].Param := 0; // G1 Linear [Op16 P1]
    Lines10[46].X := 272.896; Lines10[46].Z := 269.441; Lines10[46].F := 400; Lines10[46].CMD := 1; Lines10[46].Param := 0; // G1 Linear [Op16 P1]
    Lines10[47].X := 272.637; Lines10[47].Z := 270.418; Lines10[47].F := 400; Lines10[47].CMD := 1; Lines10[47].Param := 0; // G1 Linear [Op16 P1]
    Lines10[48].X := 272.371; Lines10[48].Z := 271.393; Lines10[48].F := 400; Lines10[48].CMD := 1; Lines10[48].Param := 0; // G1 Linear [Op16 P1]
    Lines10[49].X := 272.098; Lines10[49].Z := 272.365; Lines10[49].F := 400; Lines10[49].CMD := 1; Lines10[49].Param := 0; // G1 Linear [Op16 P1]
    Lines10[50].X := 271.889; Lines10[50].Z := 273.092; Lines10[50].F := 400; Lines10[50].CMD := 1; Lines10[50].Param := 0; // G1 Linear [Op16 P1]
    Lines10[51].X := 271.604; Lines10[51].Z := 274.060; Lines10[51].F := 400; Lines10[51].CMD := 1; Lines10[51].Param := 0; // G1 Linear [Op16 P1]
    Lines10[52].X := 271.386; Lines10[52].Z := 274.784; Lines10[52].F := 400; Lines10[52].CMD := 1; Lines10[52].Param := 0; // G1 Linear [Op16 P1]
    Lines10[53].X := 271.090; Lines10[53].Z := 275.747; Lines10[53].F := 400; Lines10[53].CMD := 1; Lines10[53].Param := 0; // G1 Linear [Op16 P1]
    Lines10[54].X := 270.863; Lines10[54].Z := 276.467; Lines10[54].F := 400; Lines10[54].CMD := 1; Lines10[54].Param := 0; // G1 Linear [Op16 P1]
    Lines10[55].X := 270.555; Lines10[55].Z := 277.426; Lines10[55].F := 400; Lines10[55].CMD := 1; Lines10[55].Param := 0; // G1 Linear [Op16 P1]
    Lines10[56].X := 270.241; Lines10[56].Z := 278.382; Lines10[56].F := 400; Lines10[56].CMD := 1; Lines10[56].Param := 0; // G1 Linear [Op16 P1]
    Lines10[57].X := 269.920; Lines10[57].Z := 279.336; Lines10[57].F := 400; Lines10[57].CMD := 1; Lines10[57].Param := 0; // G1 Linear [Op16 P1]
    Lines10[58].X := 269.592; Lines10[58].Z := 280.287; Lines10[58].F := 400; Lines10[58].CMD := 1; Lines10[58].Param := 0; // G1 Linear [Op16 P1]
    Lines10[59].X := 269.341; Lines10[59].Z := 280.998; Lines10[59].F := 400; Lines10[59].CMD := 1; Lines10[59].Param := 0; // G1 Linear [Op16 P1]
    Lines10[60].X := 269.087; Lines10[60].Z := 281.708; Lines10[60].F := 400; Lines10[60].CMD := 1; Lines10[60].Param := 0; // G1 Linear [Op16 P1]
    Lines10[61].X := 268.743; Lines10[61].Z := 282.653; Lines10[61].F := 400; Lines10[61].CMD := 1; Lines10[61].Param := 0; // G1 Linear [Op16 P1]
    Lines10[62].X := 268.480; Lines10[62].Z := 283.360; Lines10[62].F := 400; Lines10[62].CMD := 1; Lines10[62].Param := 0; // G1 Linear [Op16 P1]
    Lines10[63].X := 268.124; Lines10[63].Z := 284.300; Lines10[63].F := 400; Lines10[63].CMD := 1; Lines10[63].Param := 0; // G1 Linear [Op16 P1]
    Lines10[64].X := 267.761; Lines10[64].Z := 285.238; Lines10[64].F := 400; Lines10[64].CMD := 1; Lines10[64].Param := 0; // G1 Linear [Op16 P1]
    Lines10[65].X := 267.485; Lines10[65].Z := 285.939; Lines10[65].F := 400; Lines10[65].CMD := 1; Lines10[65].Param := 0; // G1 Linear [Op16 P1]
    Lines10[66].X := 267.204; Lines10[66].Z := 286.639; Lines10[66].F := 400; Lines10[66].CMD := 1; Lines10[66].Param := 0; // G1 Linear [Op16 P1]
    Lines10[67].X := 266.825; Lines10[67].Z := 287.570; Lines10[67].F := 400; Lines10[67].CMD := 1; Lines10[67].Param := 0; // G1 Linear [Op16 P1]
    Lines10[68].X := 266.439; Lines10[68].Z := 288.499; Lines10[68].F := 400; Lines10[68].CMD := 1; Lines10[68].Param := 0; // G1 Linear [Op16 P1]
    Lines10[69].X := 266.046; Lines10[69].Z := 289.425; Lines10[69].F := 400; Lines10[69].CMD := 1; Lines10[69].Param := 0; // G1 Linear [Op16 P1]
    Lines10[70].X := 265.747; Lines10[70].Z := 290.118; Lines10[70].F := 400; Lines10[70].CMD := 1; Lines10[70].Param := 0; // G1 Linear [Op16 P1]
    Lines10[71].X := 265.342; Lines10[71].Z := 291.040; Lines10[71].F := 400; Lines10[71].CMD := 1; Lines10[71].Param := 0; // G1 Linear [Op16 P1]
    Lines10[72].X := 265.034; Lines10[72].Z := 291.729; Lines10[72].F := 400; Lines10[72].CMD := 1; Lines10[72].Param := 0; // G1 Linear [Op16 P1]
    Lines10[73].X := 264.618; Lines10[73].Z := 292.646; Lines10[73].F := 400; Lines10[73].CMD := 1; Lines10[73].Param := 0; // G1 Linear [Op16 P1]
    Lines10[74].X := 264.302; Lines10[74].Z := 293.333; Lines10[74].F := 400; Lines10[74].CMD := 1; Lines10[74].Param := 0; // G1 Linear [Op16 P1]
    Lines10[75].X := 263.874; Lines10[75].Z := 294.245; Lines10[75].F := 400; Lines10[75].CMD := 1; Lines10[75].Param := 0; // G1 Linear [Op16 P1]
    Lines10[76].X := 263.549; Lines10[76].Z := 294.928; Lines10[76].F := 400; Lines10[76].CMD := 1; Lines10[76].Param := 0; // G1 Linear [Op16 P1]
    Lines10[77].X := 263.109; Lines10[77].Z := 295.836; Lines10[77].F := 400; Lines10[77].CMD := 1; Lines10[77].Param := 0; // G1 Linear [Op16 P1]
    Lines10[78].X := 262.663; Lines10[78].Z := 296.742; Lines10[78].F := 400; Lines10[78].CMD := 1; Lines10[78].Param := 0; // G1 Linear [Op16 P1]
    Lines10[79].X := 262.210; Lines10[79].Z := 297.645; Lines10[79].F := 400; Lines10[79].CMD := 1; Lines10[79].Param := 0; // G1 Linear [Op16 P1]
    Lines10[80].X := 261.866; Lines10[80].Z := 298.321; Lines10[80].F := 400; Lines10[80].CMD := 1; Lines10[80].Param := 0; // G1 Linear [Op16 P1]
    Lines10[81].X := 261.402; Lines10[81].Z := 299.220; Lines10[81].F := 400; Lines10[81].CMD := 1; Lines10[81].Param := 0; // G1 Linear [Op16 P1]
    Lines10[82].X := 261.049; Lines10[82].Z := 299.892; Lines10[82].F := 400; Lines10[82].CMD := 1; Lines10[82].Param := 0; // G1 Linear [Op16 P1]
    Lines10[83].X := 260.573; Lines10[83].Z := 300.786; Lines10[83].F := 400; Lines10[83].CMD := 1; Lines10[83].Param := 0; // G1 Linear [Op16 P1]
    Lines10[84].X := 260.212; Lines10[84].Z := 301.455; Lines10[84].F := 400; Lines10[84].CMD := 1; Lines10[84].Param := 0; // G1 Linear [Op16 P1]
    Lines10[85].X := 259.724; Lines10[85].Z := 302.345; Lines10[85].F := 400; Lines10[85].CMD := 1; Lines10[85].Param := 0; // G1 Linear [Op16 P1]
    Lines10[86].X := 259.229; Lines10[86].Z := 303.232; Lines10[86].F := 400; Lines10[86].CMD := 1; Lines10[86].Param := 0; // G1 Linear [Op16 P1]
    Lines10[87].X := 258.728; Lines10[87].Z := 304.117; Lines10[87].F := 400; Lines10[87].CMD := 1; Lines10[87].Param := 0; // G1 Linear [Op16 P1]
    Lines10[88].X := 258.220; Lines10[88].Z := 304.999; Lines10[88].F := 400; Lines10[88].CMD := 1; Lines10[88].Param := 0; // G1 Linear [Op16 P1]
    Lines10[89].X := 257.706; Lines10[89].Z := 305.878; Lines10[89].F := 400; Lines10[89].CMD := 1; Lines10[89].Param := 0; // G1 Linear [Op16 P1]
    Lines10[90].X := 256.790; Lines10[90].Z := 307.411; Lines10[90].F := 400; Lines10[90].CMD := 1; Lines10[90].Param := 0; // G1 Linear [Op16 P1]
    Lines10[91].X := 255.853; Lines10[91].Z := 308.937; Lines10[91].F := 400; Lines10[91].CMD := 1; Lines10[91].Param := 0; // G1 Linear [Op16 P1]
    Lines10[92].X := 254.896; Lines10[92].Z := 310.454; Lines10[92].F := 400; Lines10[92].CMD := 1; Lines10[92].Param := 0; // G1 Linear [Op16 P1]
    Lines10[93].X := 244.896; Lines10[93].Z := 300.454; Lines10[93].F := 0; Lines10[93].CMD := 0; Lines10[93].Param := 0; // G0 Rapid [Op16 P1]
    Lines10[94].X := 244.896; Lines10[94].Z := 0.000; Lines10[94].F := 0; Lines10[94].CMD := 0; Lines10[94].Param := 0; // G0 Rapid [Op16 P1]
    Lines10[95].X := 0.000; Lines10[95].Z := 0.000; Lines10[95].F := 0; Lines10[95].CMD := 0; Lines10[95].Param := 0; // G0 Rapid [Op16 P1]
    Lines10[96].X := 0.000; Lines10[96].Z := 0.000; Lines10[96].F := 0; Lines10[96].CMD := 21; Lines10[96].Param := 0; // Spindle OFF [Op16 P1]
    Lines10[97].X := 0.000; Lines10[97].Z := 0.000; Lines10[97].F := 0; Lines10[97].CMD := 21; Lines10[97].Param := 0; // Spindle OFF
    Lines10[98].X := 0.000; Lines10[98].Z := 0.000; Lines10[98].F := 0; Lines10[98].CMD := 99; Lines10[98].Param := 0; // Program END
END_DATA_BLOCK